KUKA KRL program: Calibration_7FlippedNew.src

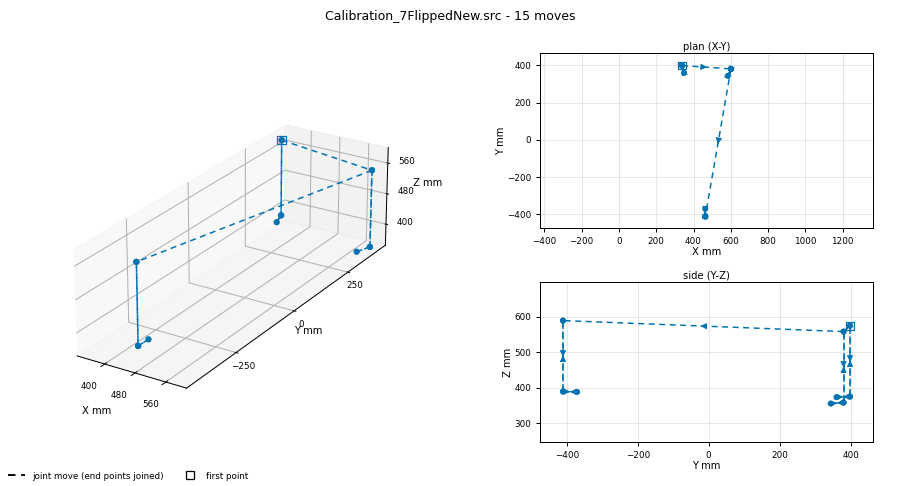
[picture p0: tool path of Calibration_7FlippedNew.src, 15 of 17 moves have a stored position in this frame; points joined in program order, loops and branches not executed]
&ACCESS RVP
&REL 1
&PARAM TEMPLATE = C:\KRC\Roboter\Template\vorgabe
&PARAM EDITMASK = *
DEF Calibration_7 ( )


;FOLD INI
;FOLD BASISTECH INI
GLOBAL INTERRUPT DECL 3 WHEN $STOPMESS==TRUE DO IR_STOPM ( )
INTERRUPT ON 3
BAS (#INITMOV,0 )
;ENDFOLD (BASISTECH INI)
;ENDFOLD (INI)

;FOLD STARTPOSITION - BASE IS 0, TOOL IS 5, SPEED IS 15%, POSITION IS A1 5,A2 -90,A3 100,A4 5,A5 -10,A6 -5,E1 0,E2 0,E3 0,E4 0
$BWDSTART = FALSE
PDAT_ACT = {VEL 15,ACC 100,APO_DIST 50}
FDAT_ACT = {TOOL_NO 5,BASE_NO 0,IPO_FRAME #BASE}
BAS (#PTP_PARAMS,15)
PTP  {A1 5,A2 -90,A3 100,A4 5,A5 -10,A6 -5,E1 0,E2 0,E3 0,E4 0}
;ENDFOLD

;FOLD LIN SPEED IS 0.1 m/sec, INTERPOLATION SETTINGS IN FOLD
$VEL.CP=0.1
$ADVANCE=3
;ENDFOLD

BAS(#VEL_PTP,10)
PTP {X 338.576, Y 398.372, Z 574.753, A -74.609, B 2.552, C 178.301, E1 0, E2 0, E3 0, E4 0, S 'B010'} C_PTP
PTP {X 338.576, Y 398.372, Z 374.752, A -74.609, B 2.552, C 178.301, E1 0, E2 0, E3 0, E4 0, S 'B010'} C_PTP
BAS(#VEL_PTP,2)
PTP {X 349.182, Y 359.844, Z 372.971, A -74.609, B 2.552, C 178.301, E1 0, E2 0, E3 0, E4 0, S 'B010'}
BAS(#VEL_PTP,10)
PTP {X 338.576, Y 398.372, Z 374.752, A -74.609, B 2.552, C 178.301, E1 0, E2 0, E3 0, E4 0, S 'B010'} C_PTP
PTP {X 338.576, Y 398.372, Z 574.753, A -74.609, B 2.552, C 178.301, E1 0, E2 0, E3 0, E4 0, S 'B010'} C_PTP
PTP {X 600.878, Y 380.066, Z 557.877, A -114.249, B 4.124, C 173.048, E1 0, E2 0, E3 0, E4 0, S 'B010'} C_PTP
PTP {X 600.878, Y 380.066, Z 357.877, A -114.249, B 4.124, C 173.048, E1 0, E2 0, E3 0, E4 0, S 'B010'} C_PTP
BAS(#VEL_PTP,2)
PTP {X 584.493, Y 343.69, Z 355, A -114.249, B 4.124, C 173.048, E1 0, E2 0, E3 0, E4 0, S 'B010'}
BAS(#VEL_PTP,10)
PTP {X 600.878, Y 380.066, Z 357.877, A -114.249, B 4.124, C 173.048, E1 0, E2 0, E3 0, E4 0, S 'B010'} C_PTP
PTP {X 600.878, Y 380.066, Z 557.877, A -114.249, B 4.124, C 173.048, E1 0, E2 0, E3 0, E4 0, S 'B010'} C_PTP
PTP {X 463.184, Y -410.69, Z 588.833, A 90.007, B 1.515, C 94.521, E1 0, E2 0, E3 0, E4 0, S 'B010'} C_PTP
PTP {X 463.184, Y -410.69, Z 388.833, A 90.007, B 1.515, C 94.521, E1 0, E2 0, E3 0, E4 0, S 'B010'} C_PTP
BAS(#VEL_PTP,2)
PTP {X 463.179, Y -370.704, Z 387.776, A 90.007, B 1.515, C 94.521, E1 0, E2 0, E3 0, E4 0, S 'B010'}
BAS(#VEL_PTP,10)
PTP {X 463.184, Y -410.69, Z 388.833, A 90.007, B 1.515, C 94.521, E1 0, E2 0, E3 0, E4 0, S 'B010'} C_PTP
PTP {X 463.184, Y -410.69, Z 588.833, A 90.007, B 1.515, C 94.521, E1 0, E2 0, E3 0, E4 0, S 'B010'} C_PTP
PTP {A1 5, A2 -90, A3 100, A4 5, A5 -10, A6 -5, E1 0, E2 0, E3 0, E4 0} C_PTP

END
